{attribute 'qualified_only'}
{attribute 'strict'}
{attribute 'to_string'}
TYPE LEDMode :
(
	Off,
	On,
	Dimmed,
	SlowFlashing,
	FastFlashing
);
END_TYPE

(* stored: Version 1.1.0.1, ProductVersion 3.1.4024.12
   DUT LEDMode: Id {ccc2dfe6-c924-4e60-8375-fc91686a2ce4} *)
